TYPE ST_EL2904 :
STRUCT
    sTerminalName       : STRING(80) := 'EL2904 | 4-Channel Safety Digital Output';
    
    // TwinSAFE physical hardware channels (Safe Outputs 1 to 4)
    bOutput             : ARRAY[1..16] OF BOOL;
    
    // Hardware status and diagnostic signals
    bError              : BOOL; // TRUE if a fault is detected (short-circuit, overload, or FSoE error)
    bReady              : BOOL; // TRUE if terminal is active and TwinSAFE communication is OK
END_STRUCT
END_TYPE

(* stored: Version 1.1.0.1
   DUT ST_EL2904: Id {b47fa1ee-8218-430d-bdaf-20385f9eef63} *)
